{attribute 'qualified_only'}
{attribute 'strict'}
TYPE eOperationMode :
(
	CurrentControlled,
	ForceControlled
);
END_TYPE

(* stored: Version 1.1.0.1, ProductVersion 3.1.4024.12
   DUT eOperationMode: Id {d213936a-7fe9-4942-aedc-46867d9c3a28} *)
